   {.imagePageWidth}
   ![LGF_DTLtoString_ISO - Aufbau der Zeichenkette nach ISO 8601](LGF_DTLtoString_ISO.png "LGF_DTLtoString_ISO - Aufbau der Zeichenkette nach ISO 8601")

   ##### Trennzeichen:

   Am Eingangsparameter `separatorDate` geben Sie das Trennzeichen zwischen den Komponenten des Kalenderdatums vor.

   ##### Beispiel:

   * separatorDate = `/` - outString = `2016/03/16…`
   * separatorDate = `-` - outString = `2016-03-16…`*/)
   END_REGION DESCRIPTION

   REGION INITIALISATION
     #tempString := '';
   END_REGION

   REGION CONVERTER
     // Set format parameters for output string
     // International ISO 8601
     // DTL  | Y| Y| Y| Y| -| M| M| -| D| D|  | H| H| :| M| M| :| S| S| .|NS|NS|NS|NS|NS|NS|NS|NS|NS
     // -----|--|--|--|--|--|--|--|--|--|--|--|--|--|--|--|--|--|--|--|--|--|--|--|--|--|--|--|--|--
     // Pos  | 1| 2| 3| 4| 5| 6| 7| 8| 9|10|11|12|13|14|15|16|17|18|19|20|21|22|23|24|25|26|27|28|29

     // Convert "Value" into "String" and place at the right position
     VAL_STRG(FORMAT := #CONVERT_FORMAT_TO_STRING,
              IN     := #date.YEAR,
              P      := #CONVERT_START_POSITION_YEAR,
              PREC   := #CONVERT_PRECISION,
              SIZE   := #CONVERT_SIZE_YEAR,
              OUT    => #tempString);    // DTL YEAR --> String --> #tempPosYear

     VAL_STRG(FORMAT := #CONVERT_FORMAT_TO_STRING,
              IN     := #date.MONTH,
              P      := #CONVERT_START_POSITION_MONTH,
              PREC   := #CONVERT_PRECISION,
              SIZE   := #CONVERT_SIZE_MONTH_DAY_HOUR_MINUTE_SECOND,
              OUT    => #tempString);     // DTL MONTH --> String --> #tempPosMonth

     VAL_STRG(FORMAT := #CONVERT_FORMAT_TO_STRING,
              IN     := #date.DAY,
              P      := #CONVERT_START_POSITION_DAY,
              PREC   := #CONVERT_PRECISION,
              SIZE   := #CONVERT_SIZE_MONTH_DAY_HOUR_MINUTE_SECOND,
              OUT    => #tempString);     // DTL DAY --> String --> #tempPosDay

     VAL_STRG(FORMAT := #CONVERT_FORMAT_TO_STRING,
              IN     := #date.HOUR,
              P      := #CONVERT_START_POSITION_HOUR,
              PREC   := #CONVERT_PRECISION,
              SIZE   := #CONVERT_SIZE_MONTH_DAY_HOUR_MINUTE_SECOND,
              OUT    => #tempString);     // DTL HOUR --> String --> #tempPosHour

     VAL_STRG(FORMAT := #CONVERT_FORMAT_TO_STRING,
              IN     := #date.MINUTE,
              P      := #CONVERT_START_POSITION_MINUTE,
              PREC   := #CONVERT_PRECISION,
              SIZE   := #CONVERT_SIZE_MONTH_DAY_HOUR_MINUTE_SECOND,
              OUT    => #tempString);     // DTL MINUTE --> String --> #tempPosMinute

     VAL_STRG(FORMAT := #CONVERT_FORMAT_TO_STRING,
              IN     := #date.SECOND,
              P      := #CONVERT_START_POSITION_SECOND,
              PREC   := #CONVERT_PRECISION,
              SIZE   := #CONVERT_SIZE_MONTH_DAY_HOUR_MINUTE_SECOND,
              OUT    => #tempString);     // DTL SECOND --> String --> #tempPosSecond

     VAL_STRG(FORMAT := #CONVERT_FORMAT_TO_STRING,
              IN     := #date.NANOSECOND,
              P      := #CONVERT_START_POSITION_NANOSECOND,
              PREC   := #CONVERT_PRECISION,
              SIZE   := #CONVERT_SIZE_NANOSECOND,
              OUT    => #tempString);     // DTL NANOSECOND --> String --> #tempPosNanosecond

     // Place separators at the right position in the string
     IF #separator = '' THEN
       #tempString[#SEPARATOR_POSITION_YEAR_MONTH] := #SEPARATOR_DATE;
       #tempString[#SEPARATOR_POSITION_MONTH_DAY] := #SEPARATOR_DATE;
     ELSE
       #tempString[#SEPARATOR_POSITION_YEAR_MONTH] := #separator;
       #tempString[#SEPARATOR_POSITION_MONTH_DAY] := #separator;
     END_IF;
     #tempString[#SEPARATOR_POSITION_HOUR_MINUTE] := #SEPARATOR_TIME;
     #tempString[#SEPARATOR_POSITION_MINUTE_SECOND] := #SEPARATOR_TIME;
     #tempString[#SEPARATOR_POSITION_SECOND_NANOSECOND] := #SEPARATOR_NANOSECOND;

     // Correcting the string, due to the conversion of a leading "0" value into a "blank".
     // Replacing of "blank" by "0"
     IF (#tempString[#CONVERT_START_POSITION_MONTH] = ' ') THEN
       #tempString[#CONVERT_START_POSITION_MONTH] := '0';
     END_IF;

     IF (#tempString[#CONVERT_START_POSITION_DAY] = ' ') THEN
       #tempString[#CONVERT_START_POSITION_DAY] := '0';
     END_IF;

     IF (#tempString[#CONVERT_START_POSITION_HOUR] = ' ') THEN
       #tempString[#CONVERT_START_POSITION_HOUR] := '0';
     END_IF;

     IF (#tempString[#CONVERT_START_POSITION_MINUTE] = ' ') THEN
       #tempString[#CONVERT_START_POSITION_MINUTE] := '0';
     END_IF;

     IF (#tempString[#CONVERT_START_POSITION_SECOND] = ' ') THEN
       #tempString[#CONVERT_START_POSITION_SECOND] := '0';
     END_IF;

     FOR #tempIndex := 0 TO #REPLACE_NANOSECOND_COUNT DO
       IF (#tempString[UINT_TO_SINT(#CONVERT_START_POSITION_NANOSECOND) + #tempIndex] = ' ') THEN
         #tempString[UINT_TO_SINT(#CONVERT_START_POSITION_NANOSECOND) + #tempIndex] := '0';
       ELSE
         EXIT;
       END_IF;
     END_FOR;
   END_REGION

   REGION OUTPUTS
     #LGF_DTLToString_ISO := #tempString;
     // no error handling needed
     ENO := TRUE;
   END_REGION
END_FUNCTION

(* ===== HMI "HMI_RT_1" =====
system functions are stored by id; their names below are inferred from use

ScreenModuleEditorView "ValueStepperInt_Vertical2" 640x480
   IOField "ioValue" at 0,48 size 80x40; FormatPattern 999999
      ProcessValue <- "value"
   Button "btnIncrease" at 0,0 size 80x40; TextOff 'Text'
      on Click: function_dd21b452("value", "delta")
   Button "btnDecrease" at 0,96 size 80x40; TextOff 'Text'
      on Click: function_b9b71300("value", "delta")
*)

(* ===== HMI "HMI_RT_5" =====
system functions are stored by id; their names below are inferred from use
connection "HMI_Connection_7": 
connection "HMI_Connection_1": ETHERNET, S7_1500_OMS

HMI tags "Template"
   "MainNavigationState" : Int, internal
   "SubNavigationState" : Int, internal
   "CurrentUserName" : WString[18], internal
   "DiagState" : Int, internal
   "PopUpBackground" : Bool, internal
   "UserName" : WString[20], internal
   "Password" : WString[20], internal
   "UserIsLoggedIn" : Bool, internal
   "CodeView" : Bool, internal
   "Brightness" : Int, internal
   "CurrentLanguage" : Bool, internal
   "CurrentRecipeName" : WString[30], internal
   "CurrentMachineState" : Int, internal
   "OptionPanelNavigationState" : Int, internal
   "ButtonDown" : Bool, internal
   "ThirdLevelNavigationState" : Int, internal
   "StartScreenName" : WString[60], internal
   "InScreenTabState" : Int, internal
   "DummyTagBool" : Bool, internal
   "DummyTagInt1" : Int, internal
   "DummyTagInt2" : Int, internal
   "DummyTagInt3" : Int, internal
   "DummyDeltaReal" : LReal, internal
   "DummTagReal1" : LReal, internal
   "DummyDeltaInt" : Int, internal

HMI tags "Filling"
   "hmiStart" : Bool = PLC GDB.hmiSignals.HMI_Start AT %DB1.DBX1006.0, 100 ms
   "hmiStop" : Bool = PLC GDB.hmiSignals.HMI_Stop AT %DB1.DBX1006.1, 100 ms
   "hmiReset" : Bool = PLC GDB.hmiSignals.HMI_Reset AT %DB1.DBX1006.2, 100 ms
   "tankLevel" : Real = PLC GDB.signals.tankSignals.actLevel AT %DB1.DBD130, 100 ms
   "tankTemperature" : Real = PLC GDB.signals.tankSignals.actTemperature AT %DB1.DBD140, 100 ms
   "tankLevelMaxReached" : Bool = PLC GDB.signals.tankSignals.maxLevel AT %DB1.DBX134.0, 100 ms
   "tankTempMax" : Bool = PLC GDB.signals.tankSignals.maxTemperature AT %DB1.DBX144.0, 100 ms
   "hmiNextBottle" : Bool = PLC GDB.hmiSignals.HMI_NextBottle AT %DB1.DBX1006.3, 100 ms
   "stateFillingTank" : Bool = PLC GDB.operate.state.FillingTank AT %DB1.DBX2.0, 100 ms
   "stateHeatingTank" : Bool = PLC GDB.operate.state.HeatingTank AT %DB1.DBX2.1, 100 ms
   "stateFillingBottle" : Bool = PLC GDB.operate.state.FillingBottle AT %DB1.DBX2.2, 100 ms
   "stateShiftingBottle" : Bool = PLC GDB.operate.state.ShiftingBottle AT %DB1.DBX2.3, 100 ms
   "stateStop" : Bool = PLC GDB.operate.state.Stop AT %DB1.DBX2.4, 100 ms
   "stateReset" : Bool = PLC GDB.operate.state.Reset AT %DB1.DBX2.5, 100 ms
   "machineState" : Int = PLC GDB.operate.machineState AT %DB1.DBW4, 100 ms
   "tankLevelMax" : Real = PLC GDB.model.tank.maxLevel AT %DB1.DBD24, 100 ms
   "stateRunning" : Bool = PLC DB_1_Sequence.statHmiStateStart, 100 ms
   "bottleID" : String[254] = PLC GDB.process.productId AT %DB1.DBX210.0, 100 ms
   "bottlesProduced" : UDInt = PLC GDB.process.numberProduced AT %DB1.DBD466, 100 ms
   "bootleNumberFaulty" : UDInt = PLC GDB.process.numberFaulty AT %DB1.DBD470, 100 ms
   "bottleLevel" : Real = PLC GDB.signals.bottleSignals.actLevel AT %DB1.DBD146, 100 ms
   "HMI_bottleLevel1" : Real, internal
   "HMI_bottleLevel2" : Real, internal
   "HMI_bottleLevel3" : Real, internal
   "HMI_bottleLevel" : Real = PLC DB_2_Filling_DB.statHmiBottleLevel AT %DB1.DBD0, 100 ms
   "HMI_doShift" : Bool = PLC DB_2_Filling_DB.statHmiDoShift AT %DB1.DBX0.0, 100 ms
      on ChangeValue: "Conveyor"()
   "qrCode" : String[254] = PLC GDB.appSignals.APP_QRCode AT %DB1.DBX1010.0, 100 ms
   "bottleFaulty" : Bool = PLC DB_2_Filling_DB.statHmiFaultyBottle AT %DB1.DBX0.0, 100 ms
   "qrCodeReceived" : Bool = PLC DB_1_Sequence.statHmiQrCodeReceived AT %DB1.DBX0.0, 100 ms
      on ChangeValue: "HandleQrCode"()
   "tempInvisibleObject" : Bool AT %DB1.DBX0.0
   "HMI_bottleInfo1" : Bool AT %DB1.DBX0.0
   "HMI_bottleInfo2" : Bool AT %DB1.DBX0.0
   "HMI_bottleInfo3" : Bool AT %DB1.DBX0.0
   "HMI_bottleInfo4" : Bool AT %DB1.DBX0.0
   "HMI_bottleInfoActive" : Bool, internal
   "energyFillingTank" : Real = PLC GDB.signals.energySignals.energyConsumptionFillingTank AT %DB1.DBD156, 100 ms
   "energyWaterFillingTank" : Real = PLC GDB.signals.energySignals.waterConsumptionFillingTank AT %DB1.DBD160, 100 ms
   "energyHeatingTank" : Real = PLC GDB.signals.energySignals.energyConsumptionHeatingTank AT %DB1.DBD164, 100 ms
   "energyFillingBottles" : Real = PLC GDB.signals.energySignals.energyConsumptionFillingBottles AT %DB1.DBD168, 100 ms
   "tankPressure" : Real = PLC GDB.signals.tankSignals.actPressure AT %DB1.DBD136, 100 ms
   "stateError" : Bool = PLC GDB.operate.state.Error AT %DB1.DBX2.6, 100 ms
   "hmiError" : Bool = PLC GDB.hmiSignals.HMI_Error AT %DB1.DBX1006.4, 100 ms
   "alarmIncoming" : Bool = PLC GDB.appSignals.APP_Alarm AT %DB1.DBX1266.2, 100 ms
   "batchID" : UDInt = PLC GDB.process.batchId AT %DB1.DBD478, 100 ms
   "energyGas" : Real = PLC GDB.signals.energySignals.gasConsumptionHeatingTank AT %DB1.DBD172, 100 ms

text list "Machine State": 0 'Undefined / Kein Job'; 1 'Production / Produktion'; 2 'Startup / Anlauf'; 3 'Paused / Pausiert'; 4 'Stopped / Gestoppt'; 5 'Shutdown / Beenden'; 6 'Undefined / UNBEKANNT'

text list "timeRange": 1 'Hours / Stunden'; 2 'Days / Tage'; 3 'Weeks / Wochen'; 4 'Months / Monate'; 5 'Years / Jahre'

text list "MachineState_Farfield": 0..1 '???'; 1 'OK'; 2 'ERROR / FEHLER'; 3 'PAUSED / HALT'

text list "Foil Types": 0..1 '120 - 1mm - Transparent'; 1 '120 - 3mm - Transparent'; 2 '240 - 1mm - Transparent'; 3 '240 - 3mm - Transparent'

text list "FunctionState": 0 'Disabled / Deaktiviert'; 1 'Enabled / Aktiviert'

text list "GroundPos": 0 'No / Nein'; 1 'Yes / Ja'

text list "State": 0 'Off / Aus'; 1 'On / An'

graphic list "DiagState": 0 'DiagOkay'; 1 'DiagWarning_1'; 2 'DiagDefault'

graphic list "DiagState_1": 0 'DiagOkay_1'; 1 'DiagWarning'; 2 'DiagDefault'

graphic list "DiagState_2": 0 'DiagOkay_1'; 1 'DiagWarning'; 2 'DiagDefault'

graphic list "DiagState_3": 0 'DiagOkay_White'; 1 'DiagWarning_White'; 2 'Circle'

graphic list "State": 0..1 'OK'; 3 'Error'

graphic list "Machine": 1 'Grafik_Verpackung_Step1_Blink-off'; 2 'Grafik_Verpackung_Step2'; 3 'Grafik_Verpackung_Blink-on'; 6..7 'Grafik_Verpackung_Step1_Blink-off'

screen "30_Diagnostics" 800x480, template "01_One_Nav_Level"
   on GenerateScreen: SetTag("MainNavigationState", 3)
   SysDiagControl "System diagnostics view_1" at 0,104 size 800x375
   GraphicView "Graphic view_2" at 0,0 size 800x480; Picture "PopUpBackground"
      Visibility <- "PopUpBackground"

screen "10_Startscreen" 800x480, template "01_One_Nav_Level"
   on GenerateScreen: "GetStartScreenName"(); SetTag("MainNavigationState", 1)
   GraphicView "Graphic view_2" at 0,0 size 800x480; Picture "PopUpBackground"
      Visibility <- "PopUpBackground"
   Button "Button_12" at 45,392 size 90x32; TextOn 'Place bottles'; TextOff 'Reset / Place bottle'
      on Press: ResetBit("hmiError")
      Visibility <- "hmiError"
   Rectangle "Rectangle_8" at 682,361 size 88x104
      Visibility <- "HMI_bottleInfoActive"
   GraphicView "Graphic view_4" at 213,87 size 249x237; Picture "Graphic_13"
   Button "Button_4" at 45,159 size 90x48; TextOff 'Start'
      on Press: SetBit("hmiStart")
      on Release: ResetBit("hmiStart")
      Appearance <- "stateRunning"
      ObjectEnable <- "stateRunning"
   Button "Button_5" at 45,215 size 90x48; TextOff 'Stop'
      on Press: SetBit("hmiStop")
      on Release: ResetBit("hmiStop")
      ObjectEnable <- "stateRunning"
      Appearance <- "stateRunning"
   Button "Button_6" at 45,271 size 90x48; TextOff 'Reset'
      on Press: SetBit("hmiReset"); ResetBit("HMI_bottleInfo1"); ResetBit("HMI_bottleInfo2"); ResetBit("HMI_bottleInfo3"); ResetBit("HMI_bottleInfo4"); ResetBit("HMI_bottleInfoActive")
      on Release: ResetBit("hmiReset")
      ObjectEnable <- "stateStop"
      Appearance <- "stateStop"
   IOField "ioKPI" at 700,269 size 68x28; FormatPattern 99.9; Unit  
      ProcessValue <- "tankTemperature"
   IOField "ioKPI_1" at 687,239 size 76x28; FormatPattern 9999
      ProcessValue <- "tankLevel"
   TextField "Text field_3" at 496,160 size 150x25; Text 'Bottles produced'
   Button "Button_1" at 45,354 size 90x32; TextOff 'Reset / Next bottle'
      on Press: SetBit("hmiNextBottle")
      on Release: ResetBit("hmiNextBottle")
      Appearance <- "stateFillingBottle"
      ObjectEnable <- "stateFillingBottle"
   TextField "Text field_1" at 610,106 size 150x25; Text 'Filling tank'
      Visibility <- "stateFillingTank"
   TextField "Text field_5" at 496,106 size 49x25; Text 'State'
   TextField "Text field_6" at 610,106 size 150x25; Text 'Heating tank'
      Visibility <- "stateHeatingTank"
   TextField "Text field_7" at 610,106 size 150x25; Text 'Filling bottle'
      Visibility <- "stateFillingBottle"
   TextField "Text field_8" at 610,106 size 150x25; Text 'Shifting bottle'
      Visibility <- "stateShiftingBottle"
   TextField "Text field_9" at 610,106 size 150x25; Text 'Stop'
      Visibility <- "stateStop"
   TextField "Text field_10" at 610,106 size 150x25; Text 'Reset'
      Visibility <- "stateReset"
   IOField "ioKPI_2" at 638,160 size 124x28; FormatPattern 9999999999
      ProcessValue <- "bottlesProduced"
   TextField "Text field_11" at 496,191 size 119x25; Text 'Bottles faulty'
   IOField "ioKPI_3" at 638,191 size 124x28; FormatPattern 9999999999
      ProcessValue <- "bootleNumberFaulty"
   IOField "ioKPI_4" at 695,329 size 68x28; FormatPattern 9.99
      ProcessValue <- "bottleLevel"
   GraphicView "Graphic view_13" at 326,321 size 17x21; Picture "Graphic_18"
   Bar "Bar_1" at 223,115 size 229x206; MinimumValue 0; MaximumValue 1600
      ProcessValue <- "tankLevel"
      Appearance <- "tankTemperature"
   GraphicView "Graphic view_7" at 617,192 size 23x23; Picture "Graphic_58"
      Visibility <- "bottleFaulty"
   Line "Line_1" at 200,422 size 266x0
      Visibility <- "bottlesProduced"
   Rectangle "Rectangle_5" at 356,418 size 32x8
      Visibility <- "bottlesProduced"
   Rectangle "Rectangle_6" at 396,418 size 32x8
      Visibility <- "bottlesProduced"
   Rectangle "Rectangle_7" at 436,418 size 32x8
      Visibility <- "bottlesProduced"
   Line "Line_2" at 200,422 size 225x0
      Visibility <- "bottlesProduced"
   Line "Line_3" at 200,422 size 185x0
      Visibility <- "bottlesProduced"
   Button "Button_2" at 322,431 size 26x22; TextOff 'Text'; PictureOff "Graphic_50"
      on Click: SetBit("HMI_bottleInfo1"); ResetBit("HMI_bottleInfo2"); ResetBit("HMI_bottleInfo3"); ResetBit("HMI_bottleInfo4"); "HandleBottleInfo"()
   Button "Button_7" at 361,431 size 26x22; TextOff 'Text'; PictureOff "Graphic_50"
      on Click: SetBit("HMI_bottleInfo2"); ResetBit("HMI_bottleInfo1"); ResetBit("HMI_bottleInfo3"); ResetBit("HMI_bottleInfo4"); "HandleBottleInfo"()
      Visibility <- "bottlesProduced"
   Button "Button_3" at 400,431 size 26x22; TextOff 'Text'; PictureOff "Graphic_50"
      on Click: SetBit("HMI_bottleInfo3"); ResetBit("HMI_bottleInfo1"); ResetBit("HMI_bottleInfo2"); ResetBit("HMI_bottleInfo4"); "HandleBottleInfo"()
      Visibility <- "bottlesProduced"
   Button "Button_8" at 440,430 size 26x22; TextOff 'Text'; PictureOff "Graphic_50"
      on Click: SetBit("HMI_bottleInfo4"); ResetBit("HMI_bottleInfo1"); ResetBit("HMI_bottleInfo2"); ResetBit("HMI_bottleInfo3"); "HandleBottleInfo"()
      Visibility <- "bottlesProduced"
   IOField "I/O field_1" at 2,459 size 20x20; FormatPattern 1
      Visibility <- "tempInvisibleObject"
      ProcessValue <- "qrCodeReceived"
   GraphicView "Graphic view_1" at 689,384 size 76x76; Picture "QRCode_bottle_one"
      Visibility <- "HMI_bottleInfo1"
   TextField "Text field_2" at 666,359 size 78x25; Text 'bottle 1'
      Visibility <- "HMI_bottleInfo1"
   TextField "Text field_12" at 665,359 size 78x25; Text 'bottle 2'
      Visibility <- "HMI_bottleInfo2"
   GraphicView "Graphic view_3" at 689,384 size 76x76; Picture "QRCode_bottle_two"
      Visibility <- "HMI_bottleInfo2"
   TextField "Text field_13" at 666,359 size 78x25; Text 'bottle 3'
      Visibility <- "HMI_bottleInfo3"
   TextField "Text field_14" at 665,359 size 78x25; Text 'bottle 4'
      Visibility <- "HMI_bottleInfo4"
   GraphicView "Graphic view_5" at 688,384 size 76x76; Picture "QRCode_bottle_three"
      Visibility <- "HMI_bottleInfo3"
   GraphicView "Graphic view_6" at 688,386 size 76x76; Picture "QRCode_bottle_four"
      Visibility <- "HMI_bottleInfo4"
   Button "Button_10" at 501,392 size 100x32; TextOff 'Energy data'; PictureOff "Graphic_50"
      on Click: function_efd93a16("EnergyInfo", 0, 0, -1, -1, 1)
   IOField "ioKPI_6" at 671,299 size 92x28; FormatPattern 999.9
      ProcessValue <- "tankPressure"
   Button "Button_11" at 45,392 size 90x32; TextOn 'Place bottles'; TextOff 'Reset / Push bottle'
      on Press: SetBit("hmiError")
      Visibility <- "hmiError"
   GraphicIOField "D6_Pilotlight_Red" at 92,109 size 40x40; PictureOn "Design_6_PilotLight_Red_On"; PictureOff "Design_6_PilotLight_Red_Off"
      ProcessValue <- "stateError"
   GraphicIOField "D6_Pilotlight_Green" at 48,109 size 40x40; PictureOn "Design_6_PilotLight_Green_On"; PictureOff "Design_6_PilotLight_Green_Off"
      ProcessValue <- "stateRunning"
   TextField "Text field_4" at 610,106 size 150x25; Text 'Error'
      Visibility <- "stateError"
   GraphicView "Graphic view_12" at 138,390 size 28x35; Picture "Graphic_73"
   GraphicView "Graphic view_14" at 138,353 size 28x35; Picture "Graphic_74"
   TextField "Text field_15" at 496,239 size 113x25; Text 'Tank level (l)'
   TextField "Text field_16" at 496,269 size 193x25; Text 'Tank temperature (°C)'
   TextField "Text field_17" at 496,299 size 174x25; Text 'Tank pressure (hPa)'
   TextField "Text field_18" at 496,329 size 124x25; Text 'Bottle level (l)'
   Button "Button_9" at 742,362 size 26x22; TextOff 'Text'; PictureOff "Graphic_68"
      on Click: ResetBit("HMI_bottleInfo1"); ResetBit("HMI_bottleInfo2"); ResetBit("HMI_bottleInfo3"); ResetBit("HMI_bottleInfo4"); ResetBit("HMI_bottleInfoActive")
      Visibility <- "HMI_bottleInfoActive"
   IOField "I/O field_2" at 23,459 size 20x20; FormatPattern 1
      Visibility <- "tempInvisibleObject"
      ProcessValue <- "alarmIncoming"
   TextField "Text field_19" at 496,132 size 74x25; Text 'Batch Id'
   IOField "ioKPI_7" at 638,132 size 124x28; FormatPattern 9999999999
      ProcessValue <- "batchID"
   GraphicView "Graphic view_8" at 318,362 size 36x43; Picture "Graphic_72"
      Visibility <- "hmiError"
   GraphicView "bottle finished 1_1" at 279,346 size 30x70; Picture "Graphic_20"
   GraphicView "bottle finished 1_2" at 239,346 size 30x70; Picture "Graphic_20"
   GraphicView "bottle finished 1_3" at 199,346 size 30x70; Picture "Graphic_20"
   GraphicView "bottle finished 1_4" at 357,346 size 30x70; Picture "Graphic_20"
      Visibility <- "bottlesProduced"
   GraphicView "bottle finished 1_5" at 397,346 size 30x70; Picture "Graphic_20"
      Visibility <- "bottlesProduced"
   GraphicView "bottle finished 1_6" at 437,346 size 30x70; Picture "Graphic_20"
      Visibility <- "bottlesProduced"
   Bar "Bar_5" at 443,372 size 20x40; MinimumValue 0.01; MaximumValue 1
      ProcessValue <- "HMI_bottleLevel3"
      Visibility <- "bottlesProduced"
   Bar "Bar_4" at 402,372 size 20x40; MinimumValue 0.01; MaximumValue 1
      ProcessValue <- "HMI_bottleLevel2"
      Visibility <- "bottlesProduced"
   Bar "Bar_3" at 362,372 size 20x40; MinimumValue 0.01; MaximumValue 1
      ProcessValue <- "HMI_bottleLevel1"
      Visibility <- "bottlesProduced"
   GraphicView "bottle finished 1" at 318,346 size 30x70; Picture "Graphic_20"
      Visibility <- "hmiError"
   Bar "Bar_2" at 324,371 size 20x40; MinimumValue 0.01; MaximumValue 1
      ProcessValue <- "bottleLevel"
      Visibility <- "hmiError"

Template "01_One_Nav_Level" 800x480
   TextField "txtTitleBar" at 16,8 size 495x32; Text 'Industrial Edge - Tank Application / Applikation'
   Button "btnStartscreen" at 0,0 size 354x45; TextOff 'Text'
      on Click: "ActivateStartScreen"()
   Rectangle "rectSystemDiagnosticsIndicator_1" at 703,0 size 48x48
      Appearance <- "alarmIncoming"
   Rectangle "rectSystemDiagnosticsIndicator" at 752,0 size 48x48
      Appearance <- "DiagState"
   GraphicIOField "gioDiagState" at 760,8 size 32x32; PictureList "DiagState_3"
      ProcessValue <- "DiagState"
   Button "btnDiagState" at 752,0 size 48x48; TextOff 'Text'
      on Click: ActivateScreen("30_Diagnostics", 0)
   TextField "Template_Text field_1" at 720,2 size 17x46; Text '!'
   Button "btnDiagState_1" at 703,0 size 48x48; TextOff 'Text'
      on Click: function_efd93a16("Alarm", 50, 100, -1, -1, 1)

PopupScreen "Template_Logon" 320x352
   on ClearScreen: ResetBit("PopUpBackground")
   on GenerateScreen: SetBit("PopUpBackground")
   TextField "Template_Text field_1" at 16,0 size 215x40; Text 'Login'
   Button "Button_2" at 16,240 size 288x40; TextOn 'LOGIN / ANMELDEN'; TextOff 'LOGIN / ANMELDEN'
      on Click: function_a9b89908("Password", "UserName"); function_efd93a16("Template_Logon", 0, 0, 0, -1, 1)
   IOField "I/O field_1" at 16,84 size 288x40; FormatPattern ??????????????????????????????
      ProcessValue <- "UserName"
   TextField "Text field_1" at 16,56 size 288x24; Text 'User Name / Name'
   IOField "I/O field_2" at 16,168 size 288x40; FormatPattern ??????????????????????????????
      ProcessValue <- "Password"
   TextField "Text field_2" at 16,140 size 288x24; Text 'Password / Passwort'
   Button "Button_1" at 16,296 size 288x40; TextOn 'CLOSE / SCHLIESSEN'; TextOff 'CLOSE / SCHLIESSEN'
      on Click: function_efd93a16("Template_Logon", 0, 0, 0, -1, 1)
      on Press: function_b14e0dd5("ButtonDown", 0)
      Appearance <- "ButtonDown"

PopupScreen "Template_Logon_Logoff" 320x352
   on ClearScreen: ResetBit("PopUpBackground")
   on GenerateScreen: SetBit("PopUpBackground")
   TextField "Template_Text field_1" at 16,0 size 215x40; Text 'Login'
   Button "Button_2" at 16,240 size 136x40; TextOn 'LOG OFF / ABMELDEN'; TextOff 'LOG OFF / ABMELDEN'
      on Click: function_f23ef4c9()
   IOField "I/O field_1" at 16,84 size 288x40; FormatPattern ??????????????????????????????
      ProcessValue <- "UserName"
   TextField "Text field_1" at 16,56 size 288x24; Text 'User Name / Name'
   IOField "I/O field_2" at 16,168 size 288x40; FormatPattern ??????????????????????????????
      ProcessValue <- "Password"
   TextField "Text field_2" at 16,140 size 288x24; Text 'Password / Passwort'
   Button "Button_1" at 16,296 size 288x40; TextOn 'CLOSE / SCHLIESSEN'; TextOff 'CLOSE / SCHLIESSEN'
      on Click: function_efd93a16("Template_Logon_Logoff", 0, 0, 0, -1, 1)
      on Press: function_b14e0dd5("ButtonDown", 0)
      Appearance <- "ButtonDown"
   Button "Button_3" at 168,240 size 136x40; TextOn 'LOGIN / ANMELDEN'; TextOff 'LOGIN / ANMELDEN'
      on Click: function_a9b89908("Password", "UserName"); function_efd93a16("Template_Logon_Logoff", 0, 0, 0, -1, 1)

PopupScreen "Template_Recipe" 700x420
   on ClearScreen: ResetBit("PopUpBackground")
   on GenerateScreen: SetBit("PopUpBackground")
   TextField "Template_Text field_1" at 14,0 size 500x40; Text 'Recipe / Rezeptur'
   Button "Button_1" at 220,364 size 260x40; TextOn 'CLOSE / SCHLIESSEN'; TextOff 'CLOSE / SCHLIESSEN'
      on Click: function_efd93a16("Template_Recipe", 0, 0, 0, -1, 1)
      on Press: function_b14e0dd5("ButtonDown", 0)
      Appearance <- "ButtonDown"
   RecipeView "Rezepturanzeige_1" at 0,40 size 698x320

PopupScreen "OptionPanel_4_Buttons" 400x328
   GraphicView "gfxOptionPanel" at 80,30 size 18x12; Picture "ManFunctions_Off"
   TextField "textOptionPanelTitle" at 108,16 size 260x40; Text 'Option Panel Title / Titel Option Panel'
   Button "btnOptionPanelClose" at 0,0 size 40x328; TextOff 'Text'; PictureOff "Jog_Forward"
      on Press: function_efd93a16("OptionPanel_4_Buttons", 0, 0, 0, 2, 2)
   Button "btnOption1" at 80,72 size 240x40; TextOn 'Option 1'; TextOff 'Option 1 / Move to Home Position'
   Button "btnOption2" at 80,128 size 240x40; TextOn 'Option 2'; TextOff 'Option 2 / Move to Home Position'
   Button "btnOption3" at 80,184 size 240x40; TextOn 'Option 3'; TextOff 'Option 3 / RESET'
   Button "btnOption4" at 80,240 size 240x40; TextOn 'Option 4'; TextOff 'Option 4 / RESET'

SlideinScreen "GraphX_Slidein_Right" 220x480
   Button "Button_1" at 0,78 size 220x60; TextOn 'Menu Item 1'; TextOff 'Startscreen / Startseite'
      on Click: ActivateScreen("10_Startscreen", 0)
      Appearance <- "MainNavigationState"
   Button "Button_3" at 0,201 size 220x60; TextOn 'Menu Item 3'; TextOff 'Diagnostics / Diagnose'
      on Click: ActivateScreen("30_Diagnostics", 0)
      Appearance <- "MainNavigationState"
   Rectangle "Rectangle_1" at 214,78 size 6x60
      Visibility <- "MainNavigationState"
   Rectangle "Rectangle_2" at 214,140 size 6x60
      Visibility <- "MainNavigationState"
   Rectangle "Rectangle_3" at 214,201 size 6x60
      Visibility <- "MainNavigationState"
   Rectangle "Rectangle_4" at 214,262 size 6x60
      Visibility <- "MainNavigationState"

PopupScreen "BottleInfo" 320x352
   on ClearScreen: ResetBit("PopUpBackground")
   on GenerateScreen: SetBit("PopUpBackground")
   TextField "Template_Text field_1" at 16,0 size 215x40; Text 'Bottle information / Login'
   IOField "I/O field_1" at 16,84 size 288x40; FormatPattern ????
      ProcessValue <- "bottleID"
   TextField "Text field_1" at 16,56 size 288x24; Text 'Production ID / Name'
   IOField "I/O field_2" at 16,168 size 288x40; FormatPattern ??????????????????????????????
      ProcessValue <- "qrCode"
   TextField "Text field_2" at 16,140 size 288x24; Text 'QR Code / Passwort'
   Button "Button_1" at 16,296 size 288x40; TextOn 'CLOSE / SCHLIESSEN'; TextOff 'CLOSE / SCHLIESSEN'
      on Click: function_efd93a16("BottleInfo", 0, 0, 0, -1, 1)
      on Press: function_b14e0dd5("ButtonDown", 0)
      Appearance <- "ButtonDown"

PopupScreen "QRCode" 320x200
   on ClearScreen: ResetBit("PopUpBackground")
   on GenerateScreen: SetBit("PopUpBackground")
   TextField "Template_Text field_1" at 16,0 size 215x40; Text 'QR Code Information / Login'
   IOField "I/O field_2" at 16,64 size 288x40; FormatPattern ??????????????????????????????
      ProcessValue <- "qrCode"
   Button "Button_1" at 16,128 size 288x40; TextOn 'CLOSE / SCHLIESSEN'; TextOff 'CLOSE / SCHLIESSEN'
      on Click: function_efd93a16("QRCode", 0, 0, 0, -1, 1); ResetBit("qrCodeReceived")
      on Press: function_b14e0dd5("ButtonDown", 0)
      Appearance <- "ButtonDown"

PopupScreen "EnergyInfo" 370x352
   on ClearScreen: ResetBit("PopUpBackground")
   on GenerateScreen: SetBit("PopUpBackground")
   IOField "I/O field_3" at 16,248 size 160x40; FormatPattern 999999.99; Unit  Wh
      ProcessValue <- "energyFillingBottles"
   TextField "Template_Text field_1" at 16,0 size 215x40; Text 'Energy consumption / Login'
   IOField "I/O field_1" at 16,103 size 160x40; FormatPattern 9999.99; Unit  Wh
      ProcessValue <- "energyFillingTank"
   TextField "Text field_1" at 16,75 size 152x24; Text 'Filling tank / Name'
   IOField "I/O field_2" at 16,176 size 160x40; FormatPattern 9999.99; Unit  Wh
      ProcessValue <- "energyHeatingTank"
   TextField "Text field_2" at 16,148 size 144x24; Text 'Heating tank / Passwort'
   Button "Button_1" at 16,304 size 344x40; TextOn 'CLOSE / SCHLIESSEN'; TextOff 'CLOSE / SCHLIESSEN'
      on Click: function_efd93a16("EnergyInfo", 0, 0, 0, -1, 1)
      on Press: function_b14e0dd5("ButtonDown", 0)
      Appearance <- "ButtonDown"
   TextField "Text field_3" at 18,220 size 144x24; Text 'Filling bottles / Passwort'
   TextField "Text field_5" at 16,48 size 104x24; Text 'Electricity / Name'
   TextField "Text field_6" at 198,72 size 56x24; Text 'Gas / Name'
   TextField "Text field_4" at 200,147 size 56x24; Text 'Water / Name'
   IOField "I/O field_4" at 200,104 size 160x40; FormatPattern 9999.99; Unit  Wh
      ProcessValue <- "energyGas"
   IOField "I/O field_5" at 200,177 size 160x40; FormatPattern 9999.99; Unit  l
      ProcessValue <- "energyWaterFillingTank"

PopupScreen "Alarm" 700x270
   AlarmView "Alarm view_1" at 5,7 size 688x196
   Button "Button_1" at 192,216 size 288x40; TextOn 'CLOSE / SCHLIESSEN'; TextOff 'CLOSE / SCHLIESSEN'
      on Click: function_efd93a16("Alarm", 0, 0, 0, -1, 1)
      on Press: function_b14e0dd5("ButtonDown", 0)
      Appearance <- "ButtonDown"

VB script "ActivateStartScreen"
   HmiRuntime.BaseScreenName = SmartTags("StartScreenName")

VB script "CheckDiagState"
   If SmartTags("@DiagnosticsIndicatorTag") = 1 Then
   	SmartTags("DiagState") = 1
   Else
   	SmartTags("DiagState") = 0
   End If

VB script "GetStartScreenName"
   SmartTags("StartScreenName") = HmiRuntime.BaseScreenName

VB script "Conveyor"
   ' ---------------- conveyor with bottles ---------------------------
   
   Dim HMI_doShift
   Set HMI_doShift = HmiRuntime.SmartTags("HMI_doShift")
   
   If HMI_doShift.Value = True Then	
   	
   	'Timer - wait to get current value from runtime
   '	Dim counter
   '	counter = 0
   '	While counter < 500
   '		counter = counter +1
   '	Wend
   
   	Dim HMI_bottleLevel
   	Dim HMI_bottleLevel1
   	Dim HMI_bottleLevel3
   	Dim HMI_bottleLevel2
   	
   	Set HMI_bottleLevel = HmiRuntime.SmartTags("HMI_bottleLevel")
   	Set HMI_bottleLevel1 = SmartTags("HMI_bottleLevel1")
   	Set HMI_bottleLevel2 = SmartTags("HMI_bottleLevel2")
   	Set HMI_bottleLevel3 = SmartTags("HMI_bottleLevel3")
   	
   	HMI_bottleLevel3.Value = HMI_bottleLevel2.Value
   	HMI_bottleLevel2.Value = HMI_bottleLevel1.Value	
   	HMI_bottleLevel1.Value = HMI_bottleLevel.Value
   
   End If

VB script "HandleQrCode"
   Dim qrCodeReceived
   Set qrCodeReceived = HmiRuntime.SmartTags("qrCodeReceived")
   
   If qrCodeReceived.Value = True Then	
   	efd93a16-2665-4b85-bcb9-25eddcb7b6f4 QRCode,0,0,$3$hmiOn$,$3$hmiAnimationOff$,$3$hmiFast$
   End If

VB script "TEMPLATE_HandleControls"
   ' ---------------- button "Next bottle" ---------------------------
   ' => if stateFillingBottle
   
   'read value from tag
   'Dim stateFillingBottle
   'Dim buttonNextBottle
   
   'Set stateFillingBottle = HmiRuntime.SmartTags("stateFillingBottle")
   'Set buttonNextBottle = SmartTags("activateButtonNextBottle")
   
   'If stateStop.Value = True And maxTemp.Value = True Then
   'If stateFillingBottle.Value = True Then
   '	buttonNextBottle.Value = True
   'Else
   '	buttonNextBottle.Value = False
   'End If

VB script "HandleBottleInfo"
   Dim HMI_bottleInfo1
   Dim HMI_bottleInfo2
   Dim HMI_bottleInfo3
   Dim HMI_bottleInfo4
   Dim HMI_bottleInfoActive
   
   Set HMI_bottleInfo1 = SmartTags("HMI_bottleInfo1")
   Set HMI_bottleInfo2 = SmartTags("HMI_bottleInfo2")
   Set HMI_bottleInfo3 = SmartTags("HMI_bottleInfo3")
   Set HMI_bottleInfo4 = SmartTags("HMI_bottleInfo4")
   Set HMI_bottleInfoActive = SmartTags("HMI_bottleInfoActive")
   
   
   If (HMI_bottleInfo1.Value = True) Or (HMI_bottleInfo2.Value = True) Or (HMI_bottleInfo3.Value = True) Or (HMI_bottleInfo4.Value = True)  Then	
   	HMI_bottleInfoActive.Value = True
   Else
   	HMI_bottleInfoActive.Value = False
   End If
*)

(* ===== HMI "MTP1500_Runtime" =====
connection "HMI_Connection_2": ETHERNET, ILRT_S7_1500_OMS

HMI tags "Filling"
   "GDB_signals_tankSignals_actLevel" : Real = PLC GDB.signals.tankSignals.actLevel AT %DB1.DBD130, T100ms
   "GDB_hmiSignals_HMI_Start" : Bool = PLC GDB.hmiSignals.HMI_Start AT %DB1.DBX1006.0, T100ms
   "GDB_hmiSignals_HMI_Stop" : Bool = PLC GDB.hmiSignals.HMI_Stop AT %DB1.DBX1006.1, T100ms
   "GDB_hmiSignals_HMI_Reset" : Bool = PLC GDB.hmiSignals.HMI_Reset AT %DB1.DBX1006.2, T100ms
   "GDB_hmiSignals_HMI_Error" : Bool = PLC GDB.hmiSignals.HMI_Error AT %DB1.DBX1006.4, T100ms
   "GDB_hmiSignals_HMI_NextBottle" : Bool = PLC GDB.hmiSignals.HMI_NextBottle AT %DB1.DBX1006.3, T100ms
   "GDB_operate_machineState" : Int = PLC GDB.operate.machineState AT %DB1.DBW4, T100ms
   "GDB_process_productId" : String[254] = PLC GDB.process.productId AT %DB1.DBX210.0, T100ms
   "GDB_process_batchId" : UDInt = PLC GDB.process.batchId AT %DB1.DBD478, T100ms
   "GDB_process_numberProduced" : UDInt = PLC GDB.process.numberProduced AT %DB1.DBD466, T100ms
   "GDB_process_numberFaulty" : UDInt = PLC GDB.process.numberFaulty AT %DB1.DBD470, T100ms
   "GDB_signals_tankSignals_actTemperature" : Real = PLC GDB.signals.tankSignals.actTemperature AT %DB1.DBD140, T100ms
   "GDB_signals_tankSignals_actPressure" : Real = PLC GDB.signals.tankSignals.actPressure AT %DB1.DBD136, T100ms
   "GDB_signals_energySignals_energyConsumptionHeatingTank" : Real = PLC GDB.signals.energySignals.energyConsumptionHeatingTank AT %DB1.DBD164, T100ms
   "GDB_signals_energySignals_energyConsumptionFillingTank" : Real = PLC GDB.signals.energySignals.energyConsumptionFillingTank AT %DB1.DBD156, T100ms
   "GDB_signals_energySignals_energyConsumptionFillingBottles" : Real = PLC GDB.signals.energySignals.energyConsumptionFillingBottles AT %DB1.DBD168, T100ms
   "GDB_signals_energySignals_waterConsumptionFillingTank" : Real = PLC GDB.signals.energySignals.waterConsumptionFillingTank AT %DB1.DBD160, T100ms
   "GDB_signals_energySignals_gasConsumptionHeatingTank" : Real = PLC GDB.signals.energySignals.gasConsumptionHeatingTank AT %DB1.DBD172, T100ms
   "GDB_process_numberGood" : UDInt = PLC GDB.process.numberGood AT %DB1.DBD474, T100ms
   "ipcEdgeUrl" : WString[254] AT %DB1.DBX0.0
   "qrCode" : USInt = PLC GDB.process.productQRCode AT %DB1.DBB996, T100ms
   "GDB_ErrorCode" : UInt = PLC GDB.signals.errorCode AT %DB1.DBW208, T100ms
   "GDB_model_bottle_AB" : Real = PLC GDB.model.bottle.AB AT %DB1.DBD44, T100ms
   "GDB_model_bottle_maxLevel" : Real = PLC GDB.model.bottle.maxLevel AT %DB1.DBD40, T100ms
   "GDB_model_cycleTime" : Real = PLC GDB.model.cycleTime AT %DB1.DBD8, T100ms
   "GDB_model_tank_AT" : Real = PLC GDB.model.tank.AT AT %DB1.DBD12, T100ms
   "GDB_model_tank_density" : Real = PLC GDB.model.tank.density AT %DB1.DBD36, T100ms
   "GDB_model_tank_H" : Real = PLC GDB.model.tank.H AT %DB1.DBD16, T100ms
   "GDB_model_tank_maxLevel" : Real = PLC GDB.model.tank.maxLevel AT %DB1.DBD24, T100ms
   "GDB_model_tank_maxTemperature" : Real = PLC GDB.model.tank.maxTemperature AT %DB1.DBD32, T100ms
   "GDB_model_tank_roomTemperature" : Real = PLC GDB.model.tank.roomTemperature AT %DB1.DBD28, T100ms
   "GDB_model_tank_Vin" : Real = PLC GDB.model.tank.Vin AT %DB1.DBD20, T100ms
   "GDB_productType" : UInt = PLC GDB.process.productTypeId AT %DB1.DBW482, T100ms
   "GDB_serialNumber" : String[254] = PLC GDB.process.productSerialNumber AT %DB1.DBX740.0, T100ms
   "GDB_signals_bottleSignals_actLevel" : Real = PLC GDB.signals.bottleSignals.actLevel AT %DB1.DBD146, T100ms
   "GDB_appSignals_ErrorSimulation" : Bool = PLC GDB.appSignals.APP_ErrorSimulation AT %DB1.DBX1266.0, T100ms
   "GDB_error_errorDuration" : Time = PLC GDB.errors.errorDuration AT %DB1.DBD1782, T100ms
   "GDB_error_errorTrigger" : Bool = PLC GDB.errors.errorTrigger AT %DB1.DBX1780.0, T100ms
   "GDB_hmiSignals_InstallFillingPump" : Bool = PLC GDB.hmiSignals.HMI_InstallFillingPump AT %DB1.DBX1006.5, T100ms
   "GDB_hmiSignals_HMI_RenewHeatingElement" : Bool = PLC GDB.hmiSignals.HMI_RenewHeatingElement AT %DB1.DBX1006.6, T100ms

HMI tags "Template"
   "Brightness" : Int, internal
   "InScreenTabState" : Int, internal
   "CurrentMachineState" : Int, internal
   "CurrentLanguage" : Int, internal
   "CurrentParameterSetName" : WString[254], internal
   "CurrentUserName" : WString[254], internal
   "Passwort" : WString[254], internal
   "CircleIndicator" : Int, internal
   "PowerState" : Int, internal
   "MachineState" : Int, internal
   "ErrorState" : Int, internal
   "TextListIndexTag" : Int, internal
   "GraphicListIndexTag" : Int, internal
   "DummyTagBool" : Bool, internal
   "DummyTagInt" : Int, internal
   "ProcessValue Signal" : Int, internal
   "Dummy_Status" : Int, internal

HMI tags "Animations"
   "bottleX" : Array [0..9] of UInt, internal
   "liquidX" : Array [0..9] of UInt, internal
   "topPosition" : Array [0..9] of UInt, internal
   "liquidLevel" : Array [0..9] of UInt, internal
   "shiftingTimer" : Int = PLC DB_1_Sequence.statShiftingTimer AT %DB1.DBW0, T100ms
   "shiftingCycle" : UInt = PLC GDB.model.bottle.shiftingCycle AT %DB1.DBW48, T100ms
   "currentX" : WString[254], internal

analog alarms
   1: 'Bottle is not under the filler. Cannot proceed with filling process. SR affected:', class Alarm, trigger "GDB_ErrorCode"
   2: 'Bottle damaged. Please change the bottle under the filler and reset to proceed.', class Alarm, trigger "GDB_ErrorCode"
   3: 'Bottle missing. Please place the bottle under the filler and reset to proceed.', class Alarm, trigger "GDB_ErrorCode"
   4: 'Wrong bottle type. Please change the bottle and reset to proceed.', class Alarm, trigger "GDB_ErrorCode"
   5: 'Conveyor does not work properly - detected wrong speed which may affect bottle positions. Please check the PLC program.', class Alarm, trigger "GDB_ErrorCode"
   6: 'Filler does not work properly - detected voltage drops. Please check the electrical connection of the pump.', class Alarm, trigger "GDB_ErrorCode"
   7: 'Bottle cannot be filled - valve can be blocked. Please check the valve.', class Alarm, trigger "GDB_ErrorCode"
   8: 'Product not supplied to the filler. Please check whether the main pump works correctly.', class Alarm, trigger "GDB_ErrorCode"
   9: 'Possible PLC error. Please check the Diagnostic tab of the HMI or open PLC webserver to check the diag. buffer.', class Alarm, trigger "GDB_ErrorCode"
   10: 'Possible PLC alarm. Please check the Messages tab of the HMI.', class Alarm, trigger "GDB_ErrorCode"
   11: 'No further information. Please contact your machine supplier.', class Alarm, trigger "GDB_ErrorCode"

text list "ErrorState": 1 'ROBOT ERROR'; 0 'NO ERROR'

text list "MachineState": 1 'Filling tank / Produktion'; 2 'Heating tank / Produktion'; 3 'Filling bottle / Produktion'; 4 'Shifting bottle / Produktion'; 5 'Stop / Beenden'; 6 'Reset / Produktion'; 7 'Machine fault'; 8 'Unknown'

text list "PowerState": 1 'Manual STOP'; 0 'ON'; 2 'Program STOP'

text list "ProductionState": 1..4 'Running / Stopped'; 5 'Stop / Execute'; 6 'Reset'; 7 'Machine error'; 8 'Unknown'

text list "State": 0 'Off / Aus'; 1 'On / EIn'

text list "SystemTextList_AllenBradleyEIPAlarmTextListCollection_1": 4096 'Connection lost on PLC side - @5%s@'; 4097 'Connection lost on HMI side - @5%s@'; 4098 'Maximum number of connections exceeded - @5%s@'; 4099 'Out of resources on PLC - @5%s@'; 4100 'Legitimation failed, invalid or missing password - @5%s@'; 4101 'Open request failed - @5%s@'; 4102 'Cannot connect to PLC - @5%s@'; 4103 'Open request could not be sent'; 4104 'root certificate expired for - @5%s@'; 4105 'PLC certificate untrusted for - @5%s@'

text list "SystemTextList_ConfigErrorAlarmTextLibrary_11": 1 'NameService configuration error: Implicit deletion. Subelement instance @6%s@ must be deleted explicitly.'; 2 'NameService configuration error: Implicit deletion. Alias/Format/Unit instance @6%s@ must be deleted explicitly.'

text list "SystemTextList_ConfigErrorAlarmTextLibrary_12": 1 'CDS cache - Cache folder cannot be created or reached: @6%s@'; 2 'LOC cache - Cache folder cannot be created or reached: @6%s@'

text list "SystemTextList_ConfigErrorAlarmTextLibrary_13": 1 'EvDpManager::cleanupDeletedDatapoint - alert handler config is deleted implicitly for deleted datapoint, @3%s@'; 2 'EvDpManager::cleanupDeletedDatapoint - alert handler config is deleted implicitly but still has overrides, @3%s@'; 3 'EvDpManager::cleanupDeletedDatapoint - default value config is deleted implicitly for deleted datapoint, @3%s@'; 4 'EvDpManager::cleanupDeletedDatapoint - default value config is deleted implicitly but still has overrides, @3%s@'; 5 'EvDpManager::cleanupDeletedDatapoint - initial value config is deleted implicitly for deleted datapoint, @3%s@'; 6 'EvDpManager::cleanupDeletedDatapoint - initial value config is deleted implicitly but still has overrides, @3%s@'; 7 'EvDpManager::cleanupDeletedDatapoint - distribution config is deleted implicitly for deleted datapoint, @3%s@'; 8 'EvDpManager::cleanupDeletedDatapoint - distribution config is deleted implicitly but still has overrides, @3%s@'; 9 'EvDpManager::cleanupDeletedDatapoint - rangeCheck config is deleted implicitly for deleted datapoint, @3%s@'; 10 'EvDpManager::cleanupDeletedDatapoint - rangeCheck config is deleted implicitly but still has overrides, @3%s@'

text list "SystemTextList_ConfigErrorAlarmTextLibrary_14": 1 'The configured data point type was deleted, but a configured type is still defined for the node type: @3%s@.'; 2 'The configured data point node type was deleted in the data point type, but a configured type is still defined for the element: @3%s@.'

text list "SystemTextList_ConfigErrorAlarmTextLibrary_15": 2 'Cycles: @6%s@ does not exist'; 3 'Alarms: @6%s@ exists already'; 4 'Tags: Address @6%s@ was rejected'; 1 'Connections: @6%s@ does not exist'; 5 'Tags: Acquisition mode @6%s@ is not supported.'; 6 'Cycles: @6%s@ was deleted but associated tags exist.'; 7 'Connections: @6%s@ was deleted but associated tags exist.'; 8 'Tags: Tag @6%s@ was rejected.'; 9 'Tags: Tag @6%s@ has an invalid value.'; 0 'Connections: Connection to @6%s@ could not be established.'; 65638 'Connections: Connection to @6%s@ could not be established.'; 65639 'Connections: @6%s@ disconnected.'; 65640 'Connections: Connection to the HMI device @6%s@ is lost.'; 65641 'Connections: Connection to the PLC @6%s@ is lost.'; 65541 'Connections: Timeout while establishing the connection to @6%s@.'; 65542 'Connections: @6%s@ faulty.'; 65543 'Connections: Connection to the HMI device disconnected. Connection @5%s@ was changed.'; 65544 'Connections: Connection to the HMI device disconnected. Driver property was changed for connection @5%s@.'

text list "SystemTextList_ConfigErrorAlarmTextLibrary_16": 1 'Connections: Lifecycle monitoring cycle must be shorter than the response time.'; 2 'Connections: Cyclic services are configured but not supported by the target device.'; 3 'Connections: Change-controlled reading is configured but not supported by the target device.'; 4 'Tags: The address @6%s@ does not exist in the PLC.'; 5 'Tags: The default conversion type for the address @6%s@ could not be determined.'; 6 'Tags: Invalid conversion type'; 7 'Cycles: Invalid conversion type. Conversion is not supported at HmiCycle.'; 4096 'Connections: Version of the address @6%s@ is not supported.'; 4097 'Connections: PROFIBUS address is not supported.'; 4098 'Connections: Softbus address is not supported.'; 4099 'Connections: Address type @6%s@ is not supported.'; 4100 'Connections: Invalid connection name @6%s@. Access point is being ignored.'; 4101 'Connections: Routing is not supported. @6%s@ is not used.'; 4102 'Connections: Routing is not supported. @6%s@ is not used.'; 4103 'Connections: Invalid IP address @6%s@'; 4104 'Connections: Invalid Named Connection @6%s@. Valid format: >VMD</>connection<'; 4105 'Connections: Invalid Named Connection @6%s@. VMD connection name is too long. Only 24 characters are permitted.'; 4106 'Connections: Invalid Named Connection @6%s@. Connection name is too long. Only 32 characters are permitted.'; 4107 'Connections: Rack number @6%s@ is outside of the permitted range (0..7)'; 4108 'Connections: Invalid Named Connection @6%s@. Rack is ignored.'; 4109 'Connections: Slot number @6%s@ is outside of the permitted range (1..32)'; 4110 'Connections: Invalid Named Connection @6%s@. Slot is ignored.'; 4111 'Connection could not be established. Maximum number of available connections (@6%s@) has been exceeded.'; 4112 'Connection aborted. No sign of life in the last @4%s@ ms.'; 4113 'Connection could not be established - @4%s@'; 4114 'Connection could not be established. The address @6%s@ cannot be used.'; 4115 'Connection could not be established. Invalid address @6%s@'; 4116 'Connection could not be established - @4%s@'

text list "SystemTextList_ConfigErrorAlarmTextLibrary_17": 1 'Connection could not be established. Application instance certificate is not configured.'; 2 'Connection could not be established. Server has rejected the client certificate. OPC UA status code @4%s@.'; 3 'Connection could not be established. Internal problem in the certificate store. OPC UA status code @4%s@'; 4 'Connection could not be established. Application instance certificate could not be loaded. OPC UA status code @5%s@'; 5 'Connection could not be established. Server has not provided a certificate. @4%s@'; 6 'Connection could not be established. Validation of server certificate has failed. OPC UA status code @4%s@.'; 7 'Connection was closed. Error during alarm synchronization. OPC UA status code @4%s@.'; 8 'Connection was closed. Alarm/event subscription has failed. The number of operations on the server has been exceeded.'; 9 'Connection was closed. Alarm/event subscription has failed. The number of alarm/event subscriptions on the server has been exceeded.'; 10 'Connection could not be established. Server reports a license problem. OPC UA status code @4%s@.'; 11 'Connection could not be established. Maximum number of server sessions has been exceeded.'; 12 'Connection could not be established. Safety configuration is inconsistent. @4%s@'; 13 'Connection could not be established. The address @4%s@ cannot be used.'; 14 'Connection could not be established. OPC UA status code @4%s@'; 15 'Connection aborted. OPC UA server was stopped.'; 16 'Connection aborted. No sign of life in the last @4%s@ ms.'; 17 'Connection was closed. OPC UA server maintenance.'; 18 'Connection could not be established. Invalid configuration of the authentication mode - @4%s@'; 19 'Connection could not be established. User could not be authenticated. OPC UA status code @4%s@'; 20 'Connection could not be established. Server does not permit anonymous connection. OPC UA status code @4%s@'; 21 'Connection could not be established. Certificate problem: Error when writing the safety-relevant data to @4%s@.'; 22 'Connection could not be established. Certificate problem: Unexpected file in the folder @4%s@ cannot be removed.'; 23 'Connection could not be established. User could not be authenticated. No user or password configured.'; 24 'Connection could not be established. Unexpected length of the server certificate. @4%s@'; 25 'Connection could not be established. @4%s@ is empty.'; 26 'Connection could not be established. @4%s@ has an unexpected format.'; 27 'Connection could not be established. Server endpoints cannot be read. OPC UA status code @4%s@'; 28 'Connection could not be established. No server endpoints were found. @4%s@'; 29 'Connection could not be established. Application instance certificate could not be found.'; 30 'Connection could not be established. Unexpected format of the certificate @4%s@.'; 31 'Connection could not be established. Unexpected format of the certificate block list @4%s@.'; 32 'Connection could not be established. User could not be authenticated. An encryption detail is invalid. @4%s@'; 34 'Connection could not be established. - The configured non-transparent redundancy mode @4%s@ is not supported.'; 101 'Tags: Address @6%s@ does not exist on the server.'; 103 'Tags: Address @6%s@ cannot be accessed.'; 104 'Tags: Acquisition mode is not supported for address @6%s@.'; 201 'Alarms: Address @6%s@ does not exist on the server.'; 202 'Alarms: Address @6%s@ cannot be used. The specified range filter is not an OPC UA Event Notifier.'; 203 'Alarms: Address @6%s@ cannot be used. The specified range filter does not exist on the server.'; 204 'Alarms: Address @6%s@ cannot be used because it is not an OPC UA event type.'; 205 'Alarms: Address @6%s@ cannot be used because the OPC UA condition type is not supported.'; 206 'Alarms: Address @6%s@ cannot be used because the event type does not exist on the server.'; 207 'Alarms: Acquisition type cannot be used for address @6%s@.'; 301 'Address @6%s@ cannot be used because the version number is missing.'; 302 'Address @6%s@ cannot be used because the version number is invalid.'; 303 'Address @6%s@ cannot be used because the number of '$' delimiters is invalid.'; 304 'Address @6%s@ cannot be used because the address type is invalid.'; 305 'Unsupported version @6%s@ of the address'; 401 'Unexpected OPC UA server response: @6%s@'

text list "SystemTextList_ConfigErrorAlarmTextLibrary_18": 1 'Messages: Invalid condition string for the alarm view @6%s@.'; 2 'Messages: Invalid status tag and bit for the alarm view @6%s@.'; 3 'Messages: Invalid control tag and bit for the alarm view @6%s@.'

text list "SystemTextList_ConfigErrorAlarmTextLibrary_19": 1 'Logs: Implicit deletion. Logging tag instance @6%s@ should be deleted but there are overloaded elements.'

text list "SystemTextList_ConfigErrorAlarmTextLibrary_20": 1 ''; 2 'Restart of the runtime is required.'; 3 'The correct storage medium must be ejected and inserted again.'

text list "SystemTextList_MitsubishiiQAlarmTextListCollection_1": 4096 'Connection lost on PLC side - @5%s@'; 4097 'Connection lost on HMI side - @5%s@'; 4098 'Maximum number of connections exceeded - @5%s@'; 4099 'Out of resources on PLC - @5%s@'; 4100 'Legitimation failed, invalid or missing password - @5%s@'; 4101 'Open request failed - @5%s@'; 4102 'Cannot connect to PLC - @5%s@'; 4103 'Open request could not be sent'; 4104 'root certificate expired for - @5%s@'; 4105 'PLC certificate untrusted for - @5%s@'

text list "SystemTextList_MitsubishiMCAlarmTextListCollection_1": 4096 'Connection lost on PLC side - @5%s@'; 4097 'Connection lost on HMI side - @5%s@'; 4098 'Maximum number of connections exceeded - @5%s@'; 4099 'Out of resources on PLC - @5%s@'; 4100 'Legitimation failed, invalid or missing password - @5%s@'; 4101 'Open request failed - @5%s@'; 4102 'Cannot connect to PLC - @5%s@'; 4103 'Open request could not be sent'; 4104 'root certificate expired for - @5%s@'; 4105 'PLC certificate untrusted for - @5%s@'

text list "SystemTextList_OmronEIPAlarmTextListCollection_1": 4096 'Connection lost on PLC side - @5%s@'; 4097 'Connection lost on HMI side - @5%s@'; 4098 'Maximum number of connections exceeded - @5%s@'; 4099 'Out of resources on PLC - @5%s@'; 4100 'Legitimation failed, invalid or missing password - @5%s@'; 4101 'Open request failed - @5%s@'; 4102 'Cannot connect to PLC - @5%s@'; 4103 'Open request could not be sent'; 4104 'root certificate expired for - @5%s@'; 4105 'PLC certificate untrusted for - @5%s@'

text list "SystemTextList_RuntimeCollaborationFailureReason_2": 0 'Unknown error (@3%s@)'; 1 'The system is not running or there is a network problem'; 2 'Runtime is not started on the target device.'; 3 'The System ID does not match the expected System ID (@3%s@)'; 4 'The Collaboration name does not match the expected Collaboration name '@3%s@''; 5 'Wrong or unknown certificate'; 6 'Revoked certificate'; 7 'The time difference is too big.'; 8 'No common supported message version'; 9 'System ID (@3%s@) already exists'; 10 'System name (@3%s@) already exists'; 11 'ID/Name in local configuration for Runtime Collaboration already exists'

text list "SystemTextList_S7PlusAlarmTextListCollection_2": 4096 'Connections: Connection to the PLC @5%s@ is lost'; 4097 'Connections: Connection to the HMI device @5%s@ is lost'; 4098 'Connections: Maximum number of connections exceeded - @5%s@'; 4099 'Out of resources on PLC - @5%s@'; 4100 'Legitimation failed, invalid or missing password - @5%s@'; 4101 'Request to open the connection failed - @5%s@'; 4102 'Connections: Cannot connect to PLC - @5%s@'; 4103 'Request to open the connection could not be sent'; 4104 'General certificate error for PLC - @5%s@'; 4105 'PLC certificate expired for PLC - @5%s@'; 4106 'PLC certificate is revoked for PLC - @5%s@'; 4107 'PLC certificate is untrustworthy. Manual trust is possible for - @5%s@'; 4108 'PLC certificate is untrustworthy. Manual trust is not possible for - @5%s@'

text list "SystemTextList_StdModbusRTUAlarmTextListCollection_1": 4096 'Connection lost on PLC side - @5%s@'; 4097 'Connection lost on HMI side - @5%s@'; 4098 'Maximum number of connections exceeded - @5%s@'; 4099 'Out of resources on PLC - @5%s@'; 4100 'Legitimation failed, invalid or missing password - @5%s@'; 4101 'Open request failed - @5%s@'; 4102 'Cannot connect to PLC - @5%s@'; 4103 'Open request could not be sent'; 4104 'root certificate expired for - @5%s@'; 4105 'PLC certificate untrusted for - @5%s@'

text list "SystemTextList_StdModbusTCPAlarmTextListCollection_1": 4096 'Connection lost on PLC side - @5%s@'; 4097 'Connection lost on HMI side - @5%s@'; 4098 'Maximum number of connections exceeded - @5%s@'; 4099 'Out of resources on PLC - @5%s@'; 4100 'Legitimation failed, invalid or missing password - @5%s@'; 4101 'Open request failed - @5%s@'; 4102 'Cannot connect to PLC - @5%s@'; 4103 'Open request could not be sent'; 4104 'root certificate expired for - @5%s@'; 4105 'PLC certificate untrusted for - @5%s@'

text list "Heating status": 2 'Heating'; 4..5 'Idle'

text list "Error mapping": 8000 'Bottle in wrong position'; 8001 'Cracked bottle detected'; 8002 'No bottle on the conveyor'; 8003 'Wrong bottle detected'; 8004 'Conveyor malfunction'; 8005 'Filler malfunction'; 8006 'Valve blocked'; 8007 'No flow in main pipe'; 8008 'Generic error - check the PLC buffer'; 8009 'Generic error - check the alarm buffer'; 8010 'Generic error - contact with the supplier'; 8011 ''

text list "SystemTextList_ConfigErrorAlarmTextLibrary_1": 1 'NameService configuration error: Implicit deletion. Subelement instance @6%s@ must be deleted explicitly.'; 2 'NameService configuration error: Implicit deletion. Alias/Format/Unit instance @6%s@ must be deleted explicitly.'

text list "SystemTextList_ConfigErrorAlarmTextLibrary_2": 1 'EvDpManager::cleanupDeletedDatapoint - alert handler config is deleted implicitly for deleted datapoint, @3%s@'; 2 'EvDpManager::cleanupDeletedDatapoint - alert handler config is deleted implicitly but still has overrides, @3%s@'; 3 'EvDpManager::cleanupDeletedDatapoint - default value config is deleted implicitly for deleted datapoint, @3%s@'; 4 'EvDpManager::cleanupDeletedDatapoint - default value config is deleted implicitly but still has overrides, @3%s@'; 5 'EvDpManager::cleanupDeletedDatapoint - initial value config is deleted implicitly for deleted datapoint, @3%s@'; 6 'EvDpManager::cleanupDeletedDatapoint - initial value config is deleted implicitly but still has overrides, @3%s@'; 7 'EvDpManager::cleanupDeletedDatapoint - distribution config is deleted implicitly for deleted datapoint, @3%s@'; 8 'EvDpManager::cleanupDeletedDatapoint - distribution config is deleted implicitly but still has overrides, @3%s@'; 9 'EvDpManager::cleanupDeletedDatapoint - rangeCheck config is deleted implicitly for deleted datapoint, @3%s@'; 10 'EvDpManager::cleanupDeletedDatapoint - rangeCheck config is deleted implicitly but still has overrides, @3%s@'

text list "SystemTextList_ConfigErrorAlarmTextLibrary_3": 1 'The configured data point type was deleted, but a configured type is still defined for the node type: @3%s@.'; 2 'The configured data point node type was deleted in the data point type, but a configured type is still defined for the element: @3%s@.'

text list "SystemTextList_ConfigErrorAlarmTextLibrary_4": 2 'Cycles: @6%s@ does not exist'; 3 'Alarms: @6%s@ exists already'; 4 'Tags: Address @6%s@ was rejected'; 1 'Connections: @6%s@ does not exist'; 5 'Tags: Acquisition mode @6%s@ is not supported.'; 6 'Cycles: @6%s@ was deleted but associated tags exist.'; 7 'Connections: @6%s@ was deleted but associated tags exist.'; 8 'Tags: Tag @6%s@ was rejected.'; 9 'Tags: Tag @6%s@ has an invalid value.'; 0 'Connections: Connection to @6%s@ could not be established.'; 65638 'Connections: Connection to @6%s@ could not be established.'; 65639 'Connections: @6%s@ disconnected.'; 65640 'Connections: Connection to the HMI device @6%s@ is lost.'; 65641 'Connections: Connection to the PLC @6%s@ is lost.'; 65541 'Connections: Timeout while establishing the connection to @6%s@.'; 65542 'Connections: @6%s@ faulty.'; 65543 'Connections: Connection to the HMI device disconnected. Connection @5%s@ was changed.'; 65544 'Connections: Connection to the HMI device disconnected. Driver property was changed for connection @5%s@.'

text list "SystemTextList_ConfigErrorAlarmTextLibrary_5": 1 'Connections: Lifecycle monitoring cycle must be shorter than the response time.'; 2 'Connections: Cyclic services are configured but not supported by the target device.'; 3 'Connections: Change-controlled reading is configured but not supported by the target device.'; 4 'Tags: The address @6%s@ does not exist in the PLC.'; 5 'Tags: The default conversion type for the address @6%s@ could not be determined.'; 6 'Tags: Invalid conversion type'; 7 'Cycles: Invalid conversion type. Conversion is not supported at HmiCycle.'; 4096 'Connections: Version of the address @6%s@ is not supported.'; 4097 'Connections: PROFIBUS address is not supported.'; 4098 'Connections: Softbus address is not supported.'; 4099 'Connections: Address type @6%s@ is not supported.'; 4100 'Connections: Invalid connection name @6%s@. Access point is being ignored.'; 4101 'Connections: Routing is not supported. @6%s@ is not used.'; 4102 'Connections: Routing is not supported. @6%s@ is not used.'; 4103 'Connections: Invalid IP address @6%s@'; 4104 'Connections: Invalid Named Connection @6%s@. Valid format: >VMD</>connection<'; 4105 'Connections: Invalid Named Connection @6%s@. VMD connection name is too long. Only 24 characters are permitted.'; 4106 'Connections: Invalid Named Connection @6%s@. Connection name is too long. Only 32 characters are permitted.'; 4107 'Connections: Rack number @6%s@ is outside of the permitted range (0..7)'; 4108 'Connections: Invalid Named Connection @6%s@. Rack is ignored.'; 4109 'Connections: Slot number @6%s@ is outside of the permitted range (1..32)'; 4110 'Connections: Invalid Named Connection @6%s@. Slot is ignored.'; 4111 'Connection could not be established. Maximum number of available connections (@6%s@) has been exceeded.'; 4112 'Connection aborted. No sign of life in the last @4%s@ ms.'; 4113 'Connection could not be established - @4%s@'; 4114 'Connection could not be established. The address @6%s@ cannot be used.'; 4115 'Connection could not be established. Invalid address @6%s@'; 4116 'Connection could not be established - @4%s@'

text list "SystemTextList_ConfigErrorAlarmTextLibrary_6": 1 'Connection could not be established. Application instance certificate is not configured.'; 2 'Connection could not be established. Server has rejected the client certificate. OPC UA status code @4%s@.'; 3 'Connection could not be established. Internal problem in the certificate store. OPC UA status code @4%s@'; 4 'Connection could not be established. Application instance certificate could not be loaded. OPC UA status code @4%s@'; 5 'Connection could not be established. Server has not provided a certificate. @4%s@'; 6 'Connection could not be established. Validation of server certificate has failed. OPC UA status code @4%s@.'; 7 'Connection was closed. Error during alarm synchronization. OPC UA status code @4%s@.'; 8 'Connection was closed. Alarm/event subscription has failed. The number of operations on the server has been exceeded.'; 9 'Connection was closed. Alarm/event subscription has failed. The number of alarm/event subscriptions on the server has been exceeded.'; 10 'Connection could not be established. Server reports a license problem. OPC UA status code @4%s@.'; 11 'Connection could not be established. Maximum number of server sessions has been exceeded.'; 12 'Connection could not be established. Safety configuration is inconsistent. @4%s@'; 13 'Connection could not be established. The address @4%s@ cannot be used.'; 14 'Connection could not be established. OPC UA status code @4%s@'; 15 'Connection aborted. OPC UA server was stopped.'; 16 'Connection aborted. No sign of life in the last @4%s@ ms.'; 17 'Connection was closed. OPC UA server maintenance.'; 18 'Connection could not be established. Invalid configuration of the authentication mode - @4%s@'; 19 'Connection could not be established. User could not be authenticated. OPC UA status code @4%s@'; 20 'Connection could not be established. Server does not permit anonymous connection. OPC UA status code @4%s@'; 21 'Connection could not be established. Certificate problem: Error when writing the safety-relevant data to @4%s@.'; 22 'Connection could not be established. Certificate problem: Unexpected file in the folder @4%s@ cannot be removed.'; 23 'Connection could not be established. User could not be authenticated. No user or password configured.'; 24 'Connection could not be established. Unexpected length of the server certificate. @4%s@'; 25 'Connection could not be established. @4%s@ is empty.'; 26 'Connection could not be established. @4%s@ has an unexpected format.'; 27 'Connection could not be established. Server endpoints cannot be read. OPC UA status code @4%s@'; 28 'Connection could not be established. No server endpoints were found. @4%s@'; 29 'Connection could not be established. Application instance certificate could not be found.'; 30 'Connection could not be established. Unexpected format of the certificate @4%s@.'; 31 'Connection could not be established. Unexpected format of the certificate block list @4%s@.'; 32 'Connection could not be established. User could not be authenticated. An encryption detail is invalid. @4%s@'; 34 'Connection could not be established. - The configured non-transparent redundancy mode @4%s@ is not supported.'; 101 'Tags: Address @6%s@ does not exist on the server.'; 103 'Tags: Address @6%s@ cannot be accessed.'; 104 'Tags: Acquisition mode is not supported for address @6%s@.'; 201 'Alarms: Address @6%s@ does not exist on the server.'; 202 'Alarms: Address @6%s@ cannot be used. The specified range filter is not an OPC UA Event Notifier.'; 203 'Alarms: Address @6%s@ cannot be used. The specified range filter does not exist on the server.'; 204 'Alarms: Address @6%s@ cannot be used because it is not an OPC UA event type.'; 205 'Alarms: Address @6%s@ cannot be used because the OPC UA condition type is not supported.'; 206 'Alarms: Address @6%s@ cannot be used because the event type does not exist on the server.'; 207 'Alarms: Acquisition type cannot be used for address @6%s@.'; 301 'Address @6%s@ cannot be used because the version number is missing.'; 302 'Address @6%s@ cannot be used because the version number is invalid.'; 303 'Address @6%s@ cannot be used because the number of '$' delimiters is invalid.'; 304 'Address @6%s@ cannot be used because the address type is invalid.'; 305 'Unsupported version @6%s@ of the address'; 401 'Unexpected OPC UA server response: @6%s@'

text list "SystemTextList_ConfigErrorAlarmTextLibrary_7": 1 'Messages: Invalid condition string for the alarm view @6%s@.'; 2 'Messages: Invalid status tag and bit for the alarm view @6%s@.'; 3 'Messages: Invalid control tag and bit for the alarm view @6%s@.'

text list "SystemTextList_ConfigErrorAlarmTextLibrary_8": 1 'Logs: Implicit deletion. Logging tag instance @6%s@ should be deleted but there are overloaded elements.'

text list "SystemTextList_ConfigErrorAlarmTextLibrary_9": 1 ''; 2 'Restart of the runtime is required.'; 3 'The correct storage medium must be ejected and inserted again.'

text list "SystemTextList_ConfigErrorAlarmTextLibrary_10": 1 'CDS cache - Cache folder cannot be created or reached: @6%s@'; 2 'LOC cache - Cache folder cannot be created or reached: @6%s@'

text list "SystemTextList_RuntimeCollaborationFailureReason_1": 0 'Unknown error (@3%s@)'; 1 'The system is not running or there is a network problem'; 2 'Runtime is not started on the target device.'; 3 'The System ID does not match the expected System ID (@3%s@)'; 4 'The Collaboration name does not match the expected Collaboration name '@3%s@''; 5 'Wrong or unknown certificate'; 6 'Revoked certificate'; 7 'The time difference is too big.'; 8 'No common supported message version'; 9 'System ID (@3%s@) already exists'; 10 'System name (@3%s@) already exists'; 11 'ID/Name in local configuration for Runtime Collaboration already exists'

text list "SystemTextList_S7PlusAlarmTextListCollection_1": 4096 'Connections: Connection to the PLC @4%s@ is lost'; 4097 'Connections: Connection to the HMI device @4%s@ is lost'; 4098 'Connections: Maximum number of connections exceeded - @4%s@'; 4099 'Out of resources on PLC - @4%s@'; 4100 'Legitimation failed, invalid or missing password - @4%s@'; 4101 'Request to open the connection failed - @4%s@'; 4102 'Connections: Cannot connect to PLC - @4%s@'; 4103 'Request to open the connection could not be sent'; 4104 'General certificate error for PLC - @4%s@'; 4105 'PLC certificate expired for PLC - @4%s@'; 4106 'PLC certificate is revoked for PLC - @4%s@'; 4107 'PLC certificate is untrustworthy. Manual trust is possible for - @4%s@'; 4108 'PLC certificate is untrustworthy. Manual trust is not possible for - @4%s@'

text list "SystemTextList_AllenBradleyEIPAlarmTextListCollection_7": 4096 'Connection lost on PLC side - @5%s@'; 4097 'Connection lost on HMI side - @5%s@'; 4098 'Maximum number of connections exceeded - @5%s@'; 4099 'Out of resources on PLC - @5%s@'; 4100 'Legitimation failed, invalid or missing password - @5%s@'; 4101 'Open request failed - @5%s@'; 4102 'Cannot connect to PLC - @5%s@'; 4103 'Open request could not be sent'; 4104 'root certificate expired for - @5%s@'; 4105 'PLC certificate untrusted for - @5%s@'

text list "SystemTextList_OmronEIPAlarmTextListCollection_6": 4096 'Connection lost on PLC side - @5%s@'; 4097 'Connection lost on HMI side - @5%s@'; 4098 'Maximum number of connections exceeded - @5%s@'; 4099 'Out of resources on PLC - @5%s@'; 4100 'Legitimation failed, invalid or missing password - @5%s@'; 4101 'Open request failed - @5%s@'; 4102 'Cannot connect to PLC - @5%s@'; 4103 'Open request could not be sent'; 4104 'root certificate expired for - @5%s@'; 4105 'PLC certificate untrusted for - @5%s@'

text list "SystemTextList_StdModbusTCPAlarmTextListCollection_5": 4096 'Connections: Connection to the PLC @5%s@ is lost'; 4097 'Connections: Connection to the HMI device @5%s@ is lost'; 4098 'Connections: Maximum number of connections exceeded - @5%s@'; 4099 'Out of resources on PLC - @5%s@'; 4100 'Legitimation failed, invalid or missing password - @5%s@'; 4101 'Request to open the connection failed - @5%s@'; 4102 'Connections: Cannot connect to PLC - @5%s@'; 4103 'Request to open the connection could not be sent'; 4104 'General certificate error for PLC - @5%s@'; 4105 'PLC certificate expired for PLC - @5%s@'; 4106 'PLC certificate is revoked for PLC - @5%s@'; 4107 'PLC certificate is untrustworthy. Manual trust is possible for - @5%s@'; 4108 'PLC certificate is untrustworthy. Manual trust is not possible for - @5%s@'

text list "SystemTextList_MitsubishiMCAlarmTextListCollection_4": 4096 'Connection lost on PLC side - @5%s@'; 4097 'Connection lost on HMI side - @5%s@'; 4098 'Maximum number of connections exceeded - @5%s@'; 4099 'Out of resources on PLC - @5%s@'; 4100 'Legitimation failed, invalid or missing password - @5%s@'; 4101 'Open request failed - @5%s@'; 4102 'Cannot connect to PLC - @5%s@'; 4103 'Open request could not be sent'; 4104 'root certificate expired for - @5%s@'; 4105 'PLC certificate untrusted for - @5%s@'

text list "SystemTextList_MitsubishiiQAlarmTextListCollection_3": 4096 'Connection lost on PLC side - @5%s@'; 4097 'Connection lost on HMI side - @5%s@'; 4098 'Maximum number of connections exceeded - @5%s@'; 4099 'Out of resources on PLC - @5%s@'; 4100 'Legitimation failed, invalid or missing password - @5%s@'; 4101 'Open request failed - @5%s@'; 4102 'Cannot connect to PLC - @5%s@'; 4103 'Open request could not be sent'; 4104 'root certificate expired for - @5%s@'; 4105 'PLC certificate untrusted for - @5%s@'

text list "SystemTextList_StdModbusRTUAlarmTextListCollection_8": 4096 'Connections: Connection to the PLC @5%s@ is lost'; 4097 'Connections: Connection to the HMI device @5%s@ is lost'; 4098 'Connections: Maximum number of connections exceeded - @5%s@'; 4099 'Out of resources on PLC - @5%s@'; 4100 'Legitimation failed, invalid or missing password - @5%s@'; 4101 'Request to open the connection failed - @5%s@'; 4102 'Connections: Cannot connect to PLC - @5%s@'; 4103 'Request to open the connection could not be sent'; 4104 'General certificate error for PLC - @5%s@'; 4105 'PLC certificate expired for PLC - @5%s@'; 4106 'PLC certificate is revoked for PLC - @5%s@'; 4107 'PLC certificate is untrustworthy. Manual trust is possible for - @5%s@'; 4108 'PLC certificate is untrustworthy. Manual trust is not possible for - @5%s@'

graphic list "ErrorState": 7 'No_1'; 0 'Yes'

graphic list "Machine": 1 'Grafik_Verpackungsmachine_Step1_Blink-off'; 2 'Grafik_Verpackungsmachine_Step2'; 3 'Grafik_Verpackungsmachine_Blink-on'; 4 'Grafik_Verpackungsmachine_Step1_Blink-off'

graphic list "MachineState": 7 'OFF'; 1..4 'On'; 5..6 'Paused'

graphic list "PowerState": 1 'OFF'; 0 'On'

graphic list "ProductionState": 1..4 'Running'; 0 'Stopped'

graphic list "State": 0..1 'NoError'; 2..3 'Error_4'

graphic list "qrCodes": 0 '0'; 1 '1'; 2 '2'; 3 '3'; 4 '4'; 5 '5'; 6 '6'; 7 '7'; 8 '8'; 9 '9'; 10 'def'
*)